TYPE Basic_MC_Reset_Status_typ : 
	STRUCT 
		Done : BOOL;
		Busy : BOOL;
	END_STRUCT
END_TYPE

(* stored: Version 1.1.0.1, ProductVersion 3.1.4024.3
   DUT Basic_MC_Reset_Status_typ: Id {4bffac6f-c8a5-0db9-335d-1a3d30560cfb} *)
